FUNCTION_BLOCK AdsHandle
VAR_INPUT
	ServerNetId			: STRING; 	(* Server AmsNetId *)
	ServerPort 			: UDINT;	(* Server port number *)
	
	remoteAccessPrefix	: STRING;
END_VAR
VAR_OUTPUT
	bBusy				: BOOL;
	err					: BOOL;
	errid				: UDINT;
	
	receiveBuffer		: ARRAY[0..100000] OF BYTE; //TCP style data buffer
	receiveStruct		: AdsData;
END_VAR
VAR	
	socket 				: AdsSocket; //only this needs initialization
	
	sendQueue			: AdsDataQueue;
	sendBufferQueue 	: DynamicQueue; //anything going into this needs to be a TcpStruct
	
	sendBuffer 			: ARRAY[0..50000] OF BYTE; //temp byte buffer to send if neccessary
	sendStruct			: AdsData;
	
	//setupStep 			: (CLOSE_CONNECTIONS, CREATE_LISTENER, ACCEPT_CONNECTION, FINISH_SETUP);
	sendDelay : TON;
END_VAR
VAR_STAT CONSTANT
	sendDelayTime : TIME := T#1S;
END_VAR

sendDelay(IN:= , PT:= sendDelayTime, Q=> , ET=> );
sendDelay.IN := TRUE;

IF sendDelay.Q THEN
	
	sendStruct := sendQueue.poll();
	IF NOT DataIsEmpty(arr := ADR(sendStruct), arrSize := SIZEOF(sendStruct)) THEN //if valid data to send	
		write(
			symbol := CONCAT(remoteAccessPrefix, 'receiveStruct'),
			data := ADR(sendStruct),
			dataSize := SIZEOF(sendStruct));
			
		sendDelay.IN := FALSE;
	END_IF
	
END_IF

METHOD clearBuffer : BOOL
VAR
	emptyReceiverStruct : AdsData;
END_VAR
//MEMSET(ADR(receiveBuffer), 0, SIZEOF(receiveBuffer));
receiveStruct := emptyReceiverStruct;
END_METHOD

METHOD close : BOOL
VAR_INPUT
END_VAR
socket.close();
END_METHOD

METHOD getHandlerName : STRING
getHandlerName := socket.remotePrgName;
END_METHOD

METHOD open : BOOL
VAR_INPUT
	localPrgName : STRING;
	localNetId : T_AmsNetId;
	localPort : T_AmsPort;
END_VAR
socket.open(localPrgName, localNetId, localPort);
END_METHOD

METHOD queueData : BOOL
VAR_INPUT
	data : REFERENCE TO AdsData;
END_VAR
//MEMCPY(ADR(temp), data.pValue, data.diSize);
sendQueue.push(data);
END_METHOD

METHOD read : BOOL
VAR_INPUT
	symbol : STRING;
	buffer : PVOID;
	symbolSize : UDINT;
END_VAR
IF NOT socket.readBusy THEN
	read := socket.read(
		symbol:= symbol,
		buffer := buffer,
		symbolSize := symbolSize);
END_IF
END_METHOD

METHOD write : BOOL
VAR_INPUT
	symbol : STRING;
	data : PVOID;
	dataSize : UDINT;
END_VAR
VAR
	timer : TON;
END_VAR
IF NOT socket.writeBusy THEN
	write := socket.write(
		symbol:= symbol,
		data := data,
		dataSize := dataSize);
END_IF
END_METHOD

END_FUNCTION_BLOCK

(* stored: Version 1.1.0.1, ProductVersion 3.1.4024.11
   POU AdsHandle: Id {c79b5cf0-ed09-4342-b586-884c09d02b1f}, SpecialFunc None
   Folder ADS: Id {397ac168-564f-4d9f-bd2b-91d65c609190}
   Method clearBuffer: Id {ae404a4f-38d0-43a0-a308-e6555817116c}
   Method close: Id {d5807612-1e45-4262-aeb7-154a271c7279}
   Method getHandlerName: Id {354f0417-2c9a-4e09-ae72-62818b581208}
   Method open: Id {ae52d3c0-e71c-41c0-8428-7c77ce14b4a2}
   Method queueData: Id {99d4bb4a-8b89-45bf-9ede-f7df289a5a64}
   Method read: Id {afad88cd-6f92-4fed-bea7-ed86de91b537}
   Method write: Id {f037acbd-cd50-42f0-bfc3-0854d3953628} *)
